KUKA KRL data list: Up22.dat

&ACCESS RVP2
&REL 35
&COMMENT VW380 Praegen
&PARAM DISKPATH = KRC:\R1\UPs
&PARAM TEMPLATE = C:\KRC\Roboter\Template\upvorgabe
&PARAM EDITMASK = Up999[1-999]
&PARAM TPVW_VERSION = 8.1.8
DEFDAT UP22
; FOLD ;%{H} %MKUKATPVW
; ENDFOLD
; interface to basic routines
 EXT  BAS (BAS_COMMAND  :IN,REAL  :IN )
; interface to VW-standard routines
EXT VW (VW_COMMAND:IN, BOOL: IN, REAL:IN, REAL:IN, REAL:IN, REAL:IN, BOOL :IN, E6POS :IN )
; interface to VW_USER - Call
EXT  VW_USER (VW_USER_CMD :IN,INT :IN,REAL  :IN,REAL  :IN,REAL  :IN,REAL  :IN,REAL  :IN,REAL  :IN,BOOL  :IN )
EXT  VW_USR_R (VW_USER_CMD :IN,INT :IN,REAL  :IN,REAL  :IN,REAL  :IN,REAL  :IN,REAL  :IN,REAL  :IN,BOOL  :IN )
EXT  IBGN (IBGN_COMMAND  :IN,BOOL  :IN,REAL  :IN,REAL  :IN,BOOL  :IN,E6POS  :OUT )
; interface select routine
EXTFCT INT  SELECT (SUBTYPE  :IN,INT  :IN,BOOL  :IN,ARI_TYP  :IN,INT  :IN,BOOL_TYP  :IN,INT  :IN,BOOL  :IN)
INT VW_NEXT_FREE = 13
INT VW_NFREE_SPS = 13
INT VW_MAX_SPS = 113
DECL VW_MPARA_TYP P1_D = {TOOL_NO 13,BASE_NO 1,VB 100,VE 0,ACC 100,TRG_TIME 0,MOVE_TYPE #PTP_MOTION}
DECL E6POS P1 = {X 1109.929, Y -646.7397, Z -1980.132, A 89.98483, B -60.00191, C -25.99505, S 2, T 42 , E1 0.0, E2 0.0, E3 0.0, E4 0.0, E5 0.0, E6 0.0}
DECL VW_MPARA_TYP P2_D = {TOOL_NO 13,BASE_NO 1,VB 100,VE 100,ACC 100,TRG_TIME 0,MOVE_TYPE #PTP_MOTION}
DECL E6POS P2 = {X 2295.985, Y -973.8008, Z -102.3522, A 103.3186, B 5.781309, C -85.72152, S 2, T 34 , E1 0.0, E2 0.0, E3 0.0, E4 0.0, E5 0.0, E6 0.0}
DECL VW_MPARA_TYP P3_D = {TOOL_NO 13,BASE_NO 1,VB 100,VE 100,ACC 100,TRG_TIME 0,MOVE_TYPE #PTP_MOTION}
DECL E6POS P3 = {X 1440.815, Y -388.3124, Z 1162.0, A 51.64873, B 40.22982, C -144.8506, S 2, T 2 , E1 0.0, E2 0.0, E3 0.0, E4 0.0, E5 0.0, E6 0.0}
DECL VW_MPARA_TYP P4_D = {TOOL_NO 13,BASE_NO 1,VB 100,VE 100,ACC 100,TRG_TIME 0,MOVE_TYPE #PTP_MOTION}
DECL E6POS P4 = {X 542.1659, Y 810.8661, Z 1011.198, A -1.650847, B 13.50753, C 164.8701, S 2, T 2 , E1 0.0, E2 0.0, E3 0.0, E4 0.0, E5 0.0, E6 0.0}
DECL VW_MPARA_TYP P5_D = {TOOL_NO 13,BASE_NO 1,VB 100,VE 100,ACC 100,TRG_TIME 0,MOVE_TYPE #PTP_MOTION}
DECL E6POS P5 = {X 1216.102, Y 800.3561, Z 932.821, A -0.2171801, B 0.3650334, C 165.0437, S 2, T 2 , E1 0.0, E2 0.0, E3 0.0, E4 0.0, E5 0.0, E6 0.0}
DECL VW_MPARA_TYP P6_D = {TOOL_NO 13,BASE_NO 1,VB 100,VE 100,ACC 100,TRG_TIME 0,MOVE_TYPE #PTP_MOTION}
DECL E6POS P6 = {X 1484.641, Y 799.3253, Z 931.1046, A -0.2171519, B 0.3651358, C 165.0437, S 2, T 2 , E1 0.0, E2 0.0, E3 0.0, E4 0.0, E5 0.0, E6 0.0}
DECL VW_MPARA_TYP P7_D = {TOOL_NO 13,BASE_NO 1,VB 100,VE 0,ACC 100,TRG_TIME 5,MOVE_TYPE #PTP_MOTION}
DECL E6POS P7 = {X 1529.121, Y 793.2112, Z 908.5637, A -0.217152, B 0.3651147, C 165.0437, S 2, T 2 , E1 0.0, E2 0.0, E3 0.0, E4 0.0, E5 0.0, E6 0.0}
DECL VW_MPARA_TYP P8_D = {TOOL_NO 13,BASE_NO 1,VB 100,VE 100,ACC 100,TRG_TIME 0,MOVE_TYPE #PTP_MOTION}
DECL E6POS P8 = {X 1484.641, Y 799.3253, Z 931.1046, A -0.2171519, B 0.3651358, C 165.0437, S 2, T 2 , E1 0.0, E2 0.0, E3 0.0, E4 0.0, E5 0.0, E6 0.0}
DECL VW_MPARA_TYP P9_D = {TOOL_NO 13,BASE_NO 1,VB 100,VE 100,ACC 100,TRG_TIME 0,MOVE_TYPE #PTP_MOTION}
DECL E6POS P9 = {X 1216.102, Y 800.3561, Z 932.821, A -0.2171801, B 0.3650334, C 165.0437, S 2, T 2 , E1 0.0, E2 0.0, E3 0.0, E4 0.0, E5 0.0, E6 0.0}
DECL VW_MPARA_TYP P10_D = {TOOL_NO 13,BASE_NO 1,VB 100,VE 100,ACC 100,TRG_TIME 0,MOVE_TYPE #PTP_MOTION}
DECL E6POS P10 = {X 542.1659, Y 810.8661, Z 1011.198, A -1.650847, B 13.50753, C 164.8701, S 2, T 2 , E1 0.0, E2 0.0, E3 0.0, E4 0.0, E5 0.0, E6 0.0}
DECL VW_MPARA_TYP P11_D = {TOOL_NO 13,BASE_NO 1,VB 100,VE 100,ACC 100,TRG_TIME 0,MOVE_TYPE #PTP_MOTION}
DECL E6POS P11 = {X 2295.985, Y -973.8008, Z -102.3522, A 103.3186, B 5.781309, C -85.72152, S 2, T 34 , E1 0.0, E2 0.0, E3 0.0, E4 0.0, E5 0.0, E6 0.0}
DECL VW_MPARA_TYP P12_D = {TOOL_NO 13,BASE_NO 1,VB 100,VE 0,ACC 100,TRG_TIME 0,MOVE_TYPE #PTP_MOTION}
DECL E6POS P12 = {X 1109.928, Y -646.7399, Z -1980.132, A 89.98482, B -60.0019, C -25.99505, S 2, T 42 , E1 0.0, E2 0.0, E3 0.0, E4 0.0, E5 0.0, E6 0.0}
ENDDAT
